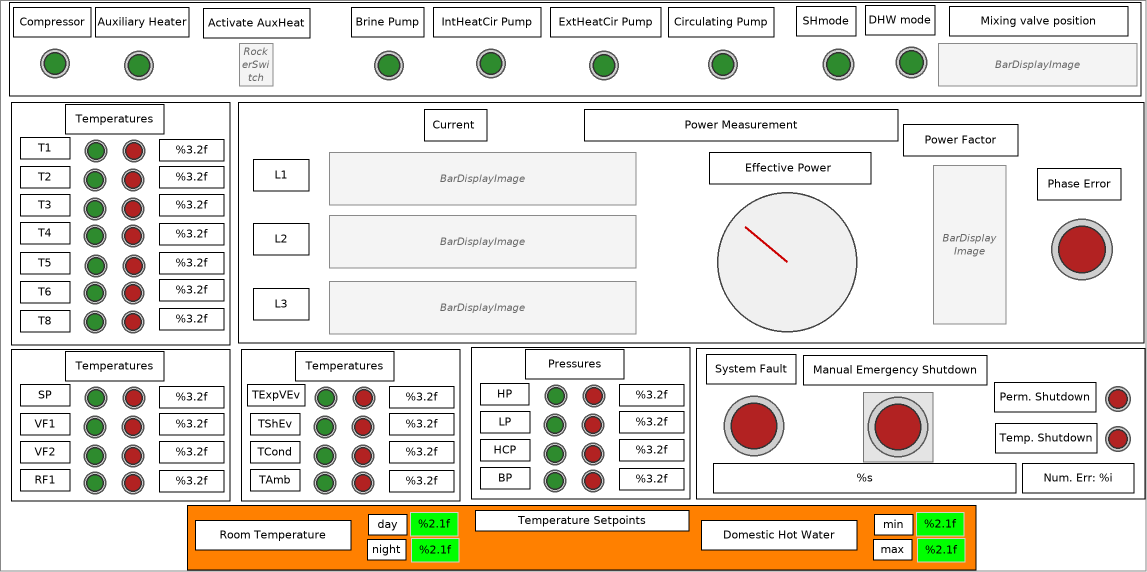
VISUALIZATION StandardVis  // 1147x572
    Group (11,102 219x243)
        Rectangle (0,0 219x243)
        Rectangle (54,2 99x30), "Temperatures"
        Rectangle (148,37 65x22), "%3.2f", text variable: Temperatures.stTempSensVR11[0].fVal
        Rectangle (148,64 65x22), "%3.2f", text variable: Temperatures.stTempSensVR11[1].fVal
        Rectangle (148,92 65x22), "%3.2f", text variable: Temperatures.stTempSensVR11[2].fVal
        Rectangle (148,121 65x22), "%3.2f", text variable: Temperatures.stTempSensVR11[3].fVal
        Rectangle (148,150 65x22), "%3.2f", text variable: Temperatures.stTempSensVR11[4].fVal
        Rectangle (148,177 65x22), "%3.2f", text variable: Temperatures.stTempSensVR11[5].fVal
        Rectangle (148,206 65x22), "%3.2f", text variable: Temperatures.stTempSensVR11[6].fVal
        Rectangle (9,35 50x22), "T1"
        Rectangle (9,64 50x22), "T2"
        Rectangle (9,92 50x22), "T3"
        Rectangle (9,120 50x22), "T4"
        Rectangle (9,150 50x22), "T5"
        Rectangle (9,179 50x22), "T6"
        Rectangle (9,208 50x22), "T8"
        Lamp1 (110,36 26x26), variable: NOT Temperatures.stTempSensVR11[0].bValid, style: Lamp-Lamp1-Red
        Lamp1 (72,36 26x26), variable: Temperatures.stTempSensVR11[0].bValid, style: Lamp-Lamp1-Green
        Lamp1 (109,65 26x26), variable: NOT Temperatures.stTempSensVR11[1].bValid, style: Lamp-Lamp1-Red
        Lamp1 (71,65 26x26), variable: Temperatures.stTempSensVR11[1].bValid, style: Lamp-Lamp1-Green
        Lamp1 (109,94 26x26), variable: NOT Temperatures.stTempSensVR11[2].bValid, style: Lamp-Lamp1-Red
        Lamp1 (71,94 26x26), variable: Temperatures.stTempSensVR11[2].bValid, style: Lamp-Lamp1-Green
        Lamp1 (109,121 26x26), variable: NOT Temperatures.stTempSensVR11[3].bValid, style: Lamp-Lamp1-Red
        Lamp1 (71,121 26x26), variable: Temperatures.stTempSensVR11[3].bValid, style: Lamp-Lamp1-Green
        Lamp1 (110,151 26x26), variable: NOT Temperatures.stTempSensVR11[4].bValid, style: Lamp-Lamp1-Red
        Lamp1 (72,151 26x26), variable: Temperatures.stTempSensVR11[4].bValid, style: Lamp-Lamp1-Green
        Lamp1 (109,178 26x26), variable: NOT Temperatures.stTempSensVR11[5].bValid, style: Lamp-Lamp1-Red
        Lamp1 (71,178 26x26), variable: Temperatures.stTempSensVR11[5].bValid, style: Lamp-Lamp1-Green
        Lamp1 (109,207 26x26), variable: NOT Temperatures.stTempSensVR11[6].bValid, style: Lamp-Lamp1-Red
        Lamp1 (71,207 26x26), variable: Temperatures.stTempSensVR11[6].bValid, style: Lamp-Lamp1-Green
    Group (11,349 219x152)
        Rectangle (0,0 219x152)
        Rectangle (54,2 99x30), "Temperatures"
        Rectangle (148,37 65x22), "%3.2f", text variable: Temperatures.stTempSensVR10[0].fVal
        Rectangle (148,64 65x22), "%3.2f", text variable: Temperatures.stTempSensVR10[1].fVal
        Rectangle (148,92 65x22), "%3.2f", text variable: Temperatures.stTempSensVR10[2].fVal
        Rectangle (148,121 65x22), "%3.2f", text variable: Temperatures.stTempSensVR10[3].fVal
        Rectangle (9,35 50x22), "SP"
        Rectangle (9,64 50x22), "VF1"
        Rectangle (9,92 50x22), "VF2"
        Rectangle (9,120 50x22), "RF1"
        Lamp1 (110,36 26x26), variable: NOT Temperatures.stTempSensVR10[0].bValid, style: Lamp-Lamp1-Red
        Lamp1 (72,36 26x26), variable: Temperatures.stTempSensVR10[0].bValid, style: Lamp-Lamp1-Green
        Lamp1 (109,65 26x26), variable: NOT Temperatures.stTempSensVR10[1].bValid, style: Lamp-Lamp1-Red
        Lamp1 (71,65 26x26), variable: Temperatures.stTempSensVR10[1].bValid, style: Lamp-Lamp1-Green
        Lamp1 (109,94 26x26), variable: NOT Temperatures.stTempSensVR10[2].bValid, style: Lamp-Lamp1-Red
        Lamp1 (71,94 26x26), variable: Temperatures.stTempSensVR10[2].bValid, style: Lamp-Lamp1-Green
        Lamp1 (109,121 26x26), variable: NOT Temperatures.stTempSensVR10[3].bValid, style: Lamp-Lamp1-Red
        Lamp1 (71,121 26x26), variable: Temperatures.stTempSensVR10[3].bValid, style: Lamp-Lamp1-Green
    Group (241,349 219x152)
        Rectangle (0,0 219x152)
        Rectangle (54,2 99x30), "Temperatures"
        Rectangle (148,37 65x22), "%3.2f", text variable: Temperatures.stTempSensPT100[0].fVal
        Rectangle (148,64 65x22), "%3.2f", text variable: Temperatures.stTempSensPT100[1].fVal
        Rectangle (148,92 65x22), "%3.2f", text variable: Temperatures.stTempSensPT100[2].fVal
        Rectangle (148,121 65x22), "%3.2f", text variable: Temperatures.stTempSensPT100[3].fVal
        Rectangle (6,35 58x22), "TExpVEv"
        Rectangle (9,64 50x22), "TShEv"
        Rectangle (9,92 50x22), "TCond"
        Rectangle (9,120 50x22), "TAmb"
        Lamp1 (110,36 26x26), variable: NOT Temperatures.stTempSensPT100[0].bValid, style: Lamp-Lamp1-Red
        Lamp1 (72,36 26x26), variable: Temperatures.stTempSensPT100[0].bValid, style: Lamp-Lamp1-Green
        Lamp1 (109,65 26x26), variable: NOT Temperatures.stTempSensPT100[1].bValid, style: Lamp-Lamp1-Red
        Lamp1 (71,65 26x26), variable: Temperatures.stTempSensPT100[1].bValid, style: Lamp-Lamp1-Green
        Lamp1 (109,94 26x26), variable: NOT Temperatures.stTempSensPT100[2].bValid, style: Lamp-Lamp1-Red
        Lamp1 (71,94 26x26), variable: Temperatures.stTempSensPT100[2].bValid, style: Lamp-Lamp1-Green
        Lamp1 (109,121 26x26), variable: NOT Temperatures.stTempSensPT100[3].bValid, style: Lamp-Lamp1-Red
        Lamp1 (71,121 26x26), variable: Temperatures.stTempSensPT100[3].bValid, style: Lamp-Lamp1-Green
    Group (471,347 219x152)
        Rectangle (0,0 219x152)
        Rectangle (54,2 99x30), "Pressures"
        Rectangle (148,37 65x22), "%3.2f", text variable: Pressures.stPress[0].fVal
        Rectangle (148,64 65x22), "%3.2f", text variable: Pressures.stPress[1].fVal
        Rectangle (148,92 65x22), "%3.2f", text variable: Pressures.stPress[2].fVal
        Rectangle (148,121 65x22), "%3.2f", text variable: Pressures.stPress[3].fVal
        Rectangle (9,36 49x22), "HP"
        Rectangle (9,64 50x22), "LP"
        Rectangle (9,92 50x22), "HCP"
        Rectangle (9,120 50x22), "BP"
        Lamp1 (110,36 26x26), variable: NOT Pressures.stPress[0].bValid, style: Lamp-Lamp1-Red
        Lamp1 (72,36 26x26), variable: Pressures.stPress[0].bValid, style: Lamp-Lamp1-Green
        Lamp1 (109,65 26x26), variable: NOT Pressures.stPress[1].bValid, style: Lamp-Lamp1-Red
        Lamp1 (71,65 26x26), variable: Pressures.stPress[1].bValid, style: Lamp-Lamp1-Green
        Lamp1 (109,94 26x26), variable: NOT Pressures.stPress[2].bValid, style: Lamp-Lamp1-Red
        Lamp1 (71,94 26x26), variable: Pressures.stPress[2].bValid, style: Lamp-Lamp1-Green
        Lamp1 (109,121 26x26), variable: NOT Pressures.stPress[3].bValid, style: Lamp-Lamp1-Red
        Lamp1 (71,121 26x26), variable: Pressures.stPress[3].bValid, style: Lamp-Lamp1-Green
    Group (238,102 906x241)
        Rectangle (0,0 906x241)
        BarDisplayImage (91,50 307x53), value: PowMeas.stPowMeas[0].fCurrent, style: BarDisplayImage-Gray, scale format: %.1f, scale 0..10
        BarDisplayImage (91,113 307x53), value: PowMeas.stPowMeas[1].fCurrent, style: BarDisplayImage-Gray, scale format: %.1f, scale 0..10
        BarDisplayImage (91,179 307x53), value: PowMeas.stPowMeas[2].fCurrent, style: BarDisplayImage-Gray, scale format: %.1f, scale 0..10
        Rectangle (15,57 56x32), "L1"
        Rectangle (15,121 56x32), "L2"
        Rectangle (15,186 56x32), "L3"
        Rectangle (346,7 314x32), "Power Measurement"
        Meter180 (421,90 256x140), value: PowMeas.fEffPow, style: Meter-Meter180-Gray, scale format: %.1f, scale 0..10
        Rectangle (471,50 162x32), "Effective Power"
        BarDisplayImage (695,63 73x159), value: PowMeas.fMeanCosPhi, style: BarDisplayImage-Gray, scale format: %.1f, scale 0.5..1
        Rectangle (665,22 115x32), "Power Factor"
        Rectangle (186,7 63x32), "Current"
        Rectangle (799,66 84x32), "Phase Error"
        Lamp1 (808,110 72x75), variable: PowMeas.bPhaseSeq, style: Lamp-Lamp1-Red
    Group (9,2 1132x94)
        Rectangle (0,0 1132x94)
        Rectangle (342,5 73x30), "Brine Pump"
        Lamp1 (29,41 34x41), variable: DigOutputs.bOutpComp, style: Lamp-Lamp1-Green
        Lamp1 (113,43 34x41), variable: DigOutputs.bOutpAH, style: Lamp-Lamp1-Green
        Rectangle (4,5 78x30), "Compressor"
        Rectangle (86,5 94x30), "Auxiliary Heater"
        Rectangle (424,5 108x30), "IntHeatCir Pump"
        Rectangle (541,5 111x30), "ExtHeatCir Pump"
        Rectangle (659,5 106x30), "Circulating Pump"
        Lamp1 (363,43 34x41), variable: StateMachine.bBrinePump, style: Lamp-Lamp1-Green
        Lamp1 (465,41 34x41), variable: StateMachine.bIntHeatCPump, style: Lamp-Lamp1-Green
        Lamp1 (578,43 34x41), variable: StateMachine.bExtHeatCPump, style: Lamp-Lamp1-Green
        Lamp1 (697,42 34x41), variable: StateMachine.bCircPump, style: Lamp-Lamp1-Green
        Lamp1 (804,44 51x37), variable: StateMachine.bSwitchVal, style: Lamp-Lamp1-Green
        Lamp1 (877,42 51x37), variable: NOT StateMachine.bSwitchVal, style: Lamp-Lamp1-Green
        Rectangle (856,3 70x30), "DHW mode"
        Rectangle (787,4 60x30), "SHmode"
        Rectangle (940,4 179x30), "Mixing valve position"
        BarDisplayImage (929,41 199x43), value: AnaOutputs.stOutpMixValv.fVal, style: BarDisplayImage-Gray, scale format: %.1f, scale 0..10
        Rectangle (194,6 107x30), "Activate AuxHeat"
        RockerSwitch (230,41 34x43), variable: StateMachine.bActAuxHeat, behaviour: TOGGLE, style: Switch-RockerSwitch-Blue
    Group (696,348 449x151)
        Rectangle (0,0 449x151)
        Rectangle (10,6 90x30), "System Fault"
        Lamp1 (23,43 70x70), variable: StateMachine.bFault, style: Lamp-Lamp1-Red
        Rectangle (107,7 184x30), "Manual Emergency Shutdown"
        PushSwitchLed (167,44 70x70), variable: StateMachine.bManEmShutdown, behaviour: TOGGLE, style: Switch-PushSwitchLed-Red
        Rectangle (17,115 303x30), "%s", text variable: StateMachine.sFaultMess, colour toggle: StateMachine.bFault
        Rectangle (298,34 102x30), "Perm. Shutdown"
        Rectangle (299,75 102x30), "Temp. Shutdown"
        Lamp1 (407,75 30x32), variable: StateMachine.bTempShut, style: Lamp-Lamp1-Red
        Lamp1 (407,35 30x32), variable: StateMachine.bPermShut, style: Lamp-Lamp1-Red
        Rectangle (326,115 112x30), "Num. Err: %i", text variable: StateMachine.nErrCount
    Group (187,505 789x65)
        Rectangle (0,0 789x65)
        Rectangle (288,5 214x21), "Temperature Setpoints"
        Rectangle (8,15 156x30), "Room Temperature"
        Textfield (223,7 48x24), "%2.1f", text variable: TempSetpoints.fRoomSetpoint, input disabled if: FALSE
            OnMouseClick: write the text variable via VisuDialogs.Numpad, min 5, max 25
        Textfield (224,33 48x24), "%2.1f", text variable: TempSetpoints.fRoomSetpointNight, input disabled if: FALSE
            OnMouseClick: write the text variable via VisuDialogs.Numpad, min 5, max 25
        Rectangle (181,9 39x21), "day"
        Rectangle (180,34 39x21), "night"
        Rectangle (514,15 156x30), "Domestic Hot Water"
        Textfield (729,7 48x24), "%2.1f", text variable: TempSetpoints.fDHWLowSP, input disabled if: FALSE
            OnMouseClick: write the text variable via VisuDialogs.Numpad, min 30, max TempSetpoints.fDHWUpSP - 1
        Textfield (730,33 48x24), "%2.1f", text variable: TempSetpoints.fDHWUpSP, input disabled if: FALSE
            OnMouseClick: write the text variable via VisuDialogs.Numpad, min TempSetpoints.fDHWLowSP + 1, max 70
        Rectangle (687,9 39x21), "min"
        Rectangle (686,34 39x21), "max"
END_VISUALIZATION

(* stored: Version 1.1.0.1, ProductVersion 3.1.4018.2
   Visu StandardVis: Id {b1795931-6c32-4978-899b-44d07e42aa57} *)
